// TwinCAT 3 PLC project VLSVacuum
// ProgramVersion: 3.1.4023.0
// libraries:
//   L2SI Vacuum Library, * (SLAC)
//   LCLS General, * (SLAC)
//   lcls-hotconnect, * (SLAC)
//   LCLSVacuumSerialDriverLib, * (SLAC)
//   PMPS, * (SLAC - LCLS)
//   Tc2_SerialCom, * (Beckhoff Automation GmbH)
//   Tc2_Standard, * (Beckhoff Automation GmbH)
//   Tc2_System, * (Beckhoff Automation GmbH)
//   Tc3_Module, * (Beckhoff Automation GmbH)
// project tree:
//   DUTs/ E_STATES.TcDUT (not stored)
//   GVLs/ GVL_Devices.TcGVL, GVL_PMPS.TcGVL, GVL_Serial.TcGVL
//   / PlcTask.TcTTO, VLSSerial.TcTTO
//   POUs/ FB_ValveBase.TcPOU (not stored), FB_VGC.TcPOU (not stored), FB_VGC_FFO.TcPOU (not stored), FB_VRC_NO.TcPOU (not stored), MAIN.TcPOU, PRG_PUMP.TcPOU, PRG_SERIAL_COM.TcPOU, PRG_VLS_VACUUM.TcPOU, PRG_VLS_WINDOW.TcPOU
// real-time tasks:
//   TASK PlcTask: cycle T#10ms, priority 20, ADS port 350
//   TASK VLSSerial: cycle T#10ms, priority 1, ADS port 351

CONFIGURATION VLSVacuum
    RESOURCE PLC ON TwinCAT3
        TASK PlcTask(INTERVAL := T#10ms, PRIORITY := 20);
        TASK VLSSerial(INTERVAL := T#10ms, PRIORITY := 1);
        PROGRAM MAIN WITH PlcTask : MAIN;
        PROGRAM PRG_SERIAL_COM WITH VLSSerial : PRG_SERIAL_COM;
    END_RESOURCE
END_CONFIGURATION

// ---- GVLs/GVL_Devices.TcGVL
VAR_GLOBAL
(*
	{attribute 'pytmc' := '
    pv: FEE:VGC:02
	'}
	FEE_VGC_02: FB_VGC;
	{attribute 'pytmc' := '
    pv: FEE:KMONO:GPI:01
	'}
	FEE_KMONO_GPI_01: FB_MKS275;
	{attribute 'pytmc' := '
    pv: FEE:KMONO:GCC:01
	'}
	FEE_KMONO_GCC_01: FB_MKS500;
	{attribute 'pytmc' := '
    pv: FEE:KMONO:PIP:01
	'}
	FEE_KMONO_PIP_01: FB_PIP_Gamma;
	{attribute 'pytmc' := '
    pv: FEE:PIP:02
	'}
	FEE_PIP_02: FB_PIP_Gamma;
	{attribute 'pytmc' := '
    pv: FEE:GPI:03
	'}
	FEE_GPI_03: FB_MKS275;
	{attribute 'pytmc' := '
    pv: FEE:GCC:03
	'}
	FEE_GCC_03: FB_MKS500;
	{attribute 'pytmc' := '
    pv: FEE:VGC:03
	'}
	FEE_VGC_03: FB_VGC_FFO;
	{attribute 'pytmc' := '
    pv: FEE:M1L:GPI:01
	'}
	FEE_M1L_GPI_01: FB_MKS275;
	{attribute 'pytmc' := '
    pv: FEE:M1L:GCC:03
	'}
	FEE_M1L_GCC_01: FB_MKS500;
	{attribute 'pytmc' := '
    pv: FEE:M1L:PIP:01
	'}
	FEE_M1L_PIP_01: FB_PIP_Gamma;
	{attribute 'pytmc' := '
    pv: FEE:PIP:03
	'}
	FEE_PIP_03: FB_PIP_Gamma;
	{attribute 'pytmc' := '
    pv: FEE:GPI:04
	'}
	FEE_GPI_04: FB_MKS275;
	{attribute 'pytmc' := '
    pv: FEE:GCC:04
	'}
	FEE_GCC_04: FB_MKS500;
	{attribute 'pytmc' := '
    pv: FEE:VGC:04
	'}
	FEE_VGC_04: FB_VGC_FFO;
	*)
END_VAR

// ---- GVLs/GVL_PMPS.TcGVL

VAR_GLOBAL
(*	
{attribute 'pytmc' := '
    pv: PLC:TST:FF1
    '}
    {attribute 'TcLinkTo' := '.q_xFastFaultOut:=TIIB[PMPS_FFO]^Channel 1^Output'}
    g_FastFaultOutput1  :   FB_HardwareFFOutput;
	
	{attribute 'pytmc' := '
    pv: PLC:TST:FF2
    '}
    {attribute 'TcLinkTo' := '.q_xFastFaultOut:=TIIB[PMPS_FFO]^Channel 2^Output'}
    g_FastFaultOutput2  :   FB_HardwareFFOutput; *)
END_VAR

// ---- GVLs/GVL_Serial.TcGVL
{attribute 'qualified_only'}
VAR_GLOBAL
	// Define COM Ports/Buffers incl. library Tc2_SerialCom
	SerialRXBuffer : ComBuffer;
	SerialTXBuffer : ComBuffer;

	// Serial Terminal
	fbSerialLineControl: SerialLineControl;
	
	//SERIAL IO
	stComIn			AT %I*	:	EL6inData22B;
	stComOut		AT %Q*	:	EL6outData22B;
	
	
	// Define COM Ports/Buffers incl. library Tc2_SerialCom
	E2_SerialRXBuffer : ComBuffer;
	E2_SerialTXBuffer : ComBuffer;
	
	// Serial Terminal
	E2_fbSerialLineControl: SerialLineControl;

	//SERIAL IO
	E2_stComIn		AT %I*	:	EL6inData22B;
	E2_stComOut		AT %Q*	:	EL6outData22B;
	
END_VAR

// ---- POUs/MAIN.TcPOU
PROGRAM MAIN
VAR
	// Variable for VLS upstream pressure bit
	{attribute 'pytmc' := '
	pv: EXT_PRESS_OK ;
	field: ZNAM NOT OK ;
	field: ONAM OK ;
	io: i ;
	'}
	bVLS_Press_OK : BOOL := FALSE; // TRUE : OK to open gate valve, FALSE : not OK to open gate valve
	
	stPTM : ST_PfeifferControl;
	fbPTM : FB_PTM_Pfeiffer;
END_VAR

(* Example main program to show how to incorporate the VLS vacuum program *)

bVLS_Press_OK := TRUE; // replace with logic for this bit, e.g. TC at vac

PRG_VLS_WINDOW(bExtPress := bVLS_Press_OK); // run the vacuum program with our interlock bit

END_PROGRAM

// ---- POUs/PRG_VLS_WINDOW.TcPOU
PROGRAM PRG_VLS_WINDOW
VAR
	xFirstPass		: BOOL;
	fbFSInit		: R_TRIG;
	
	state			: E_STATES;

	bOverride		: BOOL;
	bSetup			: BOOL;
	
	//GVL_Devices
	VGC_1			: FB_VGC;
	VGC_W			: FB_VRC_NO; // Is the Window valve NO 

	//US_GPI			: FB_MKS275;
	//US_GCC			: FB_MKS422;

	DS_GPI			: FB_MKS275;
	DS_GCC			: FB_MKS500;
END_VAR
VAR_INPUT
	bExtPress		: BOOL := FALSE; // Input for external interlock with hutch vacuum system
END_VAR

fbFSInit( CLK := TRUE, Q => xFirstPass);
(* On first PLC pass, put valve into init state*)
IF xFirstPass THEN
	state:= E_STATES.INIT;
	bOverride := FALSE;
	bSetup := FALSE;
END_IF


//STATE ACTIONS
CASE state OF

 E_STATES.INIT: 
		VGC_1.M_Set_OPN_SW(FALSE); //Isolation Valve closed
		VGC_W.M_Set_CLS_SW(FALSE); // Window valve OPEN
		VGC_1.i_xOverrideMode := VGC_W.i_xOverrideMode := FALSE;
		//Transition
		if (VGC_1.M_IsClosed() AND VGC_W.M_IsOpen()) THEN
			state:= E_STATES.NOT_SAFE;
		END_IF
		
E_STATES.NOT_SAFE: // System is not allowed to actuate, i.e all interlocks are in effect
 	VGC_1.i_xExt_OK := VGC_1.i_xEPS_OPN_OK := VGC_1.i_xEPS_CLS_OK:= FALSE; 
	VGC_W.i_xExtILK_OK:= FALSE; 
	VGC_1.i_xOverrideMode := VGC_W.i_xOverrideMode := FALSE;

	//Transition
	//IF (US_GCC.IG.xAT_VAC AND DS_GCC.IG.xAT_VAC) THEN state:= E_STATES.READY; END_IF
	IF (bExtPress AND DS_GCC.IG.xAT_VAC) THEN state:= E_STATES.READY; END_IF
	
	
	
 E_STATES.READY: // OK to MOVE
 	// Release the external interlock so the differential pressure inlk is in effect
 	VGC_1.i_xExt_OK:= VGC_1.i_xEPS_OPN_OK := VGC_1.i_xEPS_CLS_OK:= TRUE; 
	//permission to insert window valve only when US vacuum is good??
	VGC_W.i_xExtILK_OK:= bExtPress;
	// Valves  alternate positions.
	If (VGC_W.M_IsClosed()) THEN  VGC_1.M_Set_OPN_SW(TRUE);
	ELSIF (VGC_W.M_IsOpen()) THEN VGC_1.M_Set_OPN_SW(FALSE);
	END_IF
	
 
 E_STATES.OVERRIDE: 
	// Override Mode is enabled for all valves
 	VGC_1.i_xOverrideMode :=VGC_W.i_xOverrideMode := TRUE;
	// Exit of Override mode always goes back to init
 	IF NOT(bOverride) THEN state:= E_STATES.INIT; END_IF
	
	
 E_STATES.SETUP: 
	// Window valve remains retracted
 	VGC_W.i_xExtILK_OK := FALSE; 
	// Isolation valves operates like standard gate valves 
	VGC_1.i_xExt_OK := TRUE;
	// exit to init just to be safe?
	IF NOT(bSetup) THEN state:= E_STATES.INIT; END_IF
END_CASE


// STATE TRANSITIONS
// the system can go to setup state from any other state except override
IF (bSetup) AND (state<>E_STATES.OVERRIDE) THEN state:= E_STATES.SETUP; 
// the system can go to override state from any other state except setup
ELSIF (bOverride) AND (state<>E_STATES.SETUP) THEN state:= E_STATES.OVERRIDE;
//Loss of at vac signal makes the system go to init/not safe to move state
ELSIF (NOT bExtPress) OR (NOT DS_GCC.IG.xAT_VAC) THEN state:= E_STATES.INIT;
//ELSIF (NOT US_GCC.IG.xAT_VAC) OR (NOT DS_GCC.IG.xAT_VAC) THEN state:= E_STATES.INIT;
END_IF 


// Instantiate function blocks
//US_GPI(PG=>);
//US_GCC(PG:=US_GPI.PG);
DS_GPI(PG=>);
DS_GCC(PG:=DS_GPI.PG);

VGC_1(
	i_stUSG:= ,
	//i_stUSG:= US_GCC.IG,
	i_stDSG:= DS_GCC.IG , 
	i_xDis_DPIlk:= FALSE, 
	i_xEPS_OPN_OK:= , 
	i_xEPS_CLS_OK:= ,
	i_xPMPS_OK:= , 
	i_xExt_OK:= , 
	i_xOverrideMode:= , 
	i_xReset:= , 
	iq_stValve=>);

VGC_W(i_xExtILK_OK:= , 
	i_xOverrideMode:= ,
    iq_stValve=> );

END_PROGRAM

// ---- POUs/PRG_SERIAL_COM.TcPOU
PROGRAM PRG_SERIAL_COM
VAR
END_VAR

(*Instanitate Serial port com function *) 
fbSerialLineControl(
	Mode:= SERIALLINEMODE_EL6_22B,
	pComIn:= ADR(stComIn),
	pComOut:=ADR(stComOut),
	SizeComIn:= SIZEOF(stComIn),
	TxBuffer:= SerialRXBuffer,
	RxBuffer:= SerialTXBuffer,
	Error=> ,
	ErrorID=> );

END_PROGRAM

// ---- POUs/PRG_PUMP.TcPOU
PROGRAM PRG_PUMP
VAR
	{attribute 'pytmc' := '
    pv: PTM:01
	'}
	PTM_01 :  FB_PTM_Pfeiffer;
	
	// They share the same serial port
	st_Pfeiffer_CTRL 			: ARRAY[1..20] OF ST_PfeifferControl;
	st_Pfeiffer_RBK 			: ARRAY[1..20] OF ST_PfeifferStatus;
	
	fb_PfeifferCom : FB_PFEIFFER_COM;
END_VAR



//Pfeiffer Turbo

(*Assign adresses to the pfeiffer controllers connected to this serial terminal*)
st_Pfeiffer_CTRL[1].iSerialAddress :=1;
st_Pfeiffer_CTRL[1].xEnableComm := TRUE;
	
(* Instanitate the Function block for serial communication with Pfeiffer*)	
fb_PfeifferCom(astPfeifferControl := st_Pfeiffer_CTRL,
			   astPfeifferStatus:= st_Pfeiffer_RBK,
				SerialRXBuffer:= E2_SerialRXBuffer,
				SerialTXBuffer:= E2_SerialTXBuffer);
				

(* Copy Status Pv's into the PTM structure*)
PTM_01.M_Serial_IO(st_Pfeiffer_CTRL[1],st_Pfeiffer_RBK[1]);

END_PROGRAM

// ---- POUs/PRG_VLS_VACUUM.TcPOU
PROGRAM PRG_VLS_VACUUM
VAR
	stPTM : ST_PfeifferControl;
	fbPTM : FB_PTM_Pfeiffer;
END_VAR
VAR_INPUT
	bVLS_Ext_Press : BOOL := FALSE; // external interlock bit for window control
END_VAR

// VLS Vacuum Logic
PRG_VLS_WINDOW(bExtPress := bVLS_Ext_Press); // run the vacuum program with interlock bit

// VLS Pump
PRG_PUMP();

END_PROGRAM
